Fanuc KAREL source: kb00188.KL

PROGRAM KB00188
%STACKSIZE=65535
%PRIORITY=65535
%NOLOCKGROUP
VAR
P1 : STRING[80]
RESULT : INTEGER
BEGIN
P1='A'
-- UNRESOLVED_PC line 8 opcodes [27 22 2A 76 23] marker_code=14
END KB00188
